{attribute addProperty BoxType "EL6688-0000-0016"}
{attribute addProperty Id "Sync_ModeAT %I*BYTE812Control_value_update_toggleAT %I*BOOL8115Time_stamp_update_toggleAT %I*BOOL8115External_device_not_connectedAT %I*BOOL8116"}
{attribute addProperty CRC "994112877"}
{attribute addProperty SizeInBites "32"}
{attribute addProperty SizeInBytes "4"}
TYPE SYNC_Inputs_3B40F56D :
STRUCT
	{attribute addProperty Name "Sync_Mode"}
	Sync_Mode AT %I* : BYTE;
	{attribute addProperty Name "Control_value_update_toggle"}
	Control_value_update_toggle AT %I* : BOOL;
	{attribute addProperty Name "Time_stamp_update_toggle"}
	Time_stamp_update_toggle AT %I* : BOOL;
	{attribute addProperty Name "External_device_not_connected"}
	External_device_not_connected AT %I* : BOOL;
END_STRUCT
END_TYPE

(* stored: Version 1.2.0.0, ProductVersion 3.1.4024.9
   DUT SYNC_Inputs_3B40F56D: Id {70eb49b1-eb5f-4887-abf1-d38211f69560} *)
